PROGRAM Axis05_Status
VAR
//System_Bit
	Always_ON	:	BOOL	:=TRUE	;//상시 ON 
	Always_OFF	:	BOOL	:=FALSE	;//상시 OFF
	Axis05_Status_01: MC_ReadStatus;
	Axis05_Position_Read_01: MC_ReadActualPosition;
	Axis05_Velocity_Read_01: MC_ReadActualVelocity;
	Axis05_Reset_01: MC_Reset;
	Axis05_Stop_01: MC_Stop;
END_VAR

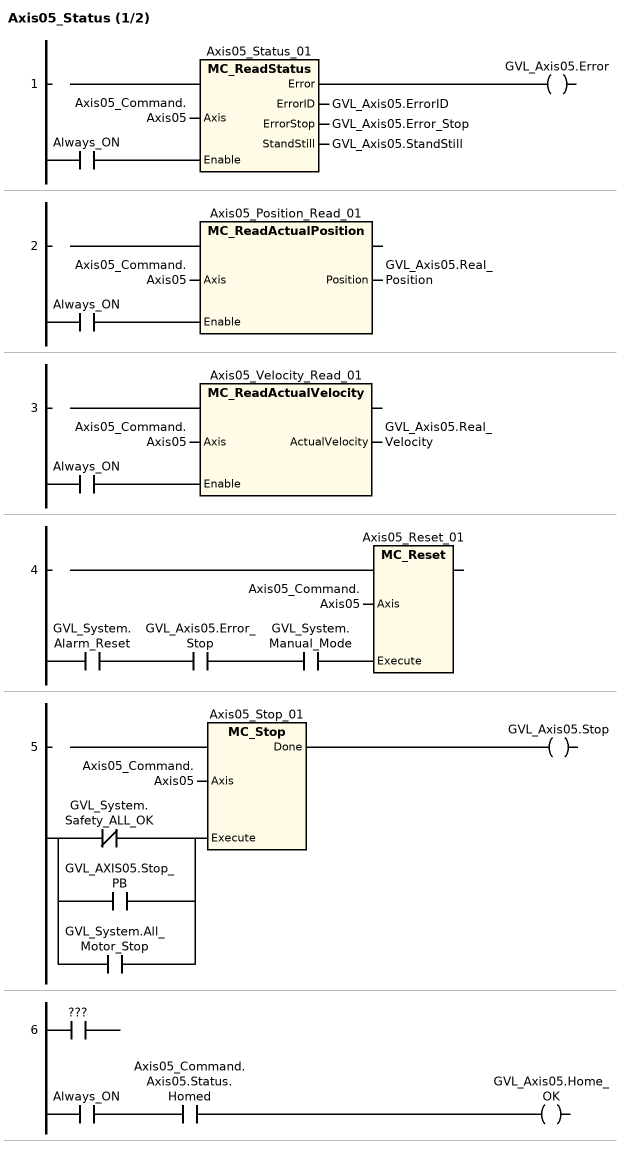
// NETWORK 1
Axis05_Status_01(
    Axis := Axis05_Command.Axis05,
    Enable := Always_ON,
    Error => GVL_Axis05.Error,
    ErrorID => GVL_Axis05.ErrorID,
    ErrorStop => GVL_Axis05.Error_Stop,
    StandStill => GVL_Axis05.StandStill); // MC_ReadStatus

// NETWORK 2
Axis05_Position_Read_01(
    Axis := Axis05_Command.Axis05,
    Enable := Always_ON,
    Position => GVL_Axis05.Real_Position); // MC_ReadActualPosition

// NETWORK 3
Axis05_Velocity_Read_01(
    Axis := Axis05_Command.Axis05,
    Enable := Always_ON,
    ActualVelocity => GVL_Axis05.Real_Velocity); // MC_ReadActualVelocity

// NETWORK 4
Axis05_Reset_01(Axis := Axis05_Command.Axis05, Execute := GVL_System.Alarm_Reset AND GVL_Axis05.Error_Stop AND GVL_System.Manual_Mode); // MC_Reset

// NETWORK 5
Axis05_Stop_01(Axis := Axis05_Command.Axis05, Execute := NOT GVL_System.Safety_ALL_OK OR GVL_AXIS05.Stop_PB OR GVL_System.All_Motor_Stop); // MC_Stop
GVL_Axis05.Stop := Axis05_Stop_01.Done;

// NETWORK 6
GVL_Axis05.Home_OK := Always_ON AND Axis05_Command.Axis05.Status.Homed;

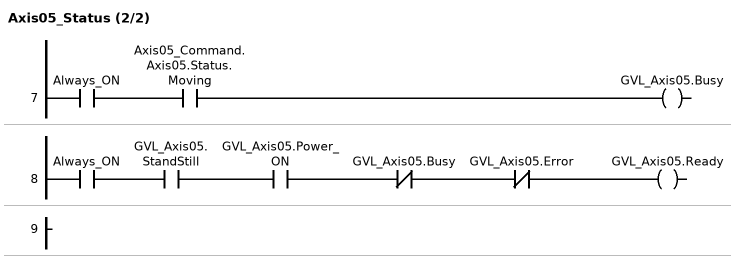
// NETWORK 7
GVL_Axis05.Busy := Always_ON AND Axis05_Command.Axis05.Status.Moving;

// NETWORK 8
GVL_Axis05.Ready := Always_ON AND GVL_Axis05.StandStill AND GVL_Axis05.Power_ON AND NOT GVL_Axis05.Busy AND NOT GVL_Axis05.Error;

// NETWORK 9

END_PROGRAM

(* stored: Version 1.1.0.1, ProductVersion 3.1.4024.15
   POU Axis05_Status: Id {cfc680cf-dda7-423e-9182-aaaf7d5606b2}, SpecialFunc None *)
